FUNCTION_BLOCK MUX_2 (* multiplexer *)
  (* Standard: 61131-3; Classification: standard selection function; Description: Copyright (c) 2013 TU Wien ACIN This program and the accompanying materials are made available under the terms of the Eclipse Public License 2.0 which is available at https://www.eclipse.org/legal/epl-2.0/ SPDX-License-Identifier: EPL-2.0 *)
  (* Version 1.0, 2013-08-30, Monika Wenger, TU Wien ACIN *)
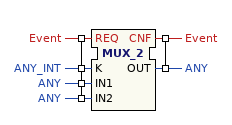
  EVENT_INPUT
    REQ WITH IN1, IN2, K; (* Service Request *)
  END_EVENT
  EVENT_OUTPUT
    CNF WITH OUT; (* Confirmation of Requested Service *)
  END_EVENT
  VAR_INPUT
    K : ANY_INT; (* Select one of n inputs *)
    IN1 : ANY; (* Input value 1 *)
    IN2 : ANY; (* Input value 2 *)
  END_VAR
  VAR_OUTPUT
    OUT : ANY; (* IN1 for K = 0, IN2 for K = 1 *)
  END_VAR
END_FUNCTION_BLOCK
